TYPE ST_Base :
STRUCT
END_STRUCT
END_TYPE

(* stored: Version 1.1.0.1, ProductVersion 3.1.4024.11
   DUT ST_Base: Id {32302bc6-943b-46d4-93d5-fada66380ce5} *)
